FUNCTION_BLOCK Flipsign
  (* Standard: 61499-2 *)
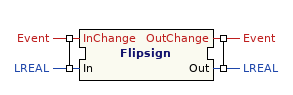
  EVENT_INPUT
    InChange WITH In;
  END_EVENT
  EVENT_OUTPUT
    OutChange WITH Out;
  END_EVENT
  VAR_INPUT
    In : LREAL;
  END_VAR
  VAR_OUTPUT
    Out : LREAL;
  END_VAR
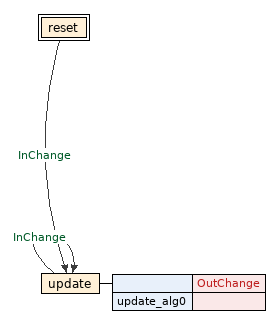
  EC_STATES
    reset;
    update : -> OutChange, update_alg0;
  END_STATES
  EC_TRANSITIONS
    reset TO update := InChange;
    update TO update := InChange;
  END_TRANSITIONS
  ALGORITHM update_alg0 IN ST:
Out := -1 * In;
  END_ALGORITHM
END_FUNCTION_BLOCK
